// TIA Portal V16 export
// export: Created 2026-06-18T12:28:25.1716274Z, ExportSetting WithDefaults, DisplayName Totally Integrated Automation Portal, DisplayVersion V16 Update 8, DisplayName TIA Portal Version Control Interface, DisplayVersion V16 Update 8, DisplayName TIA Portal Openness, DisplayVersion V16 Update 8, DisplayName STEP 7 Professional, DisplayVersion V16 Update 8, DisplayName STEP 7 Safety, DisplayVersion V16 Update 7, DisplayName WinCC Professional, DisplayVersion V16 Update 8
Screen "Motor_Control"  800x480, Number=1
  ScreenLayer 
    IOField "IO_Speed" at 192,260 size 150x44  DataFormat=Decimal, FormatPattern=9999999, Mode=InOutput
    Button "BTN_Start" at 186,170 size 124x50  Mode=Text, TextOff="启动", TextOn="启动"
    Button "BTN_Reset" at 490,170 size 124x50  Mode=Text, TextOff="复位", TextOn="复位"
    Button "BTN_Stop" at 338,170 size 124x50  Mode=Text, TextOff="停止", TextOn="停止"
    SymbolicIOField "SIO_Mode" at 512,260 size 150x44  CountVisibleItems=3, Mode=InOutput, OnValue=1, TextOff="0", TextOn="1"
    Circle "LMP_Run" at 250,85 size 48x48
    Circle "LMP_Fault" at 480,85 size 48x48
    TextField "TXT_Title" at 200,20 size 400x36  Text="电机控制画面"
    TextField "TXT_ModeLabel" at 420,260 size 80x44  Text="运行模式"
    TextField "TXT_SpeedLabel" at 120,260 size 60x44  Text="转速"
